FUNCTION FC_InitAlarmTexts : BOOL
VAR_INPUT
END_VAR
VAR
END_VAR

HMI_Texts.AlarmTexts[EAlarms.none] := 'unspecified';
HMI_Texts.AlarmTexts[EAlarms.initialized] := 'the application is initialized';
HMI_Texts.AlarmTexts[EAlarms.did_execute] := 'the component executed';
HMI_Texts.AlarmTexts[EAlarms.stopped] := 'all operations stopped';
HMI_Texts.AlarmTexts[EAlarms.stopping] := 'finishing all Control Primitives';
HMI_Texts.AlarmTexts[EAlarms.aborting] := 'aborting all Control Primitives';

HMI_Texts.AlarmTexts[ESpecialAlarmIds.recovery_request] := 'a recovery was requested; stopping operations';
HMI_Texts.AlarmTexts[ESpecialAlarmIds.definition_request] := 'a definition was requested';
HMI_Texts.AlarmTexts[ESpecialAlarmIds.strategy_received] := 'starting new strategy';
HMI_Texts.AlarmTexts[ESpecialAlarmIds.interlock_violated] := 'interlock violated';

END_FUNCTION

(* stored: Version 1.1.0.1
   POU FC_InitAlarmTexts: Id {4ec44118-7e62-4a62-8dc8-b544699bf45d}, SpecialFunc None *)
